GLOBALCONSTANTS byteconst (* Global constants *)
  (* Standard: 61499-1 *)
  (* Version 1.0, 2024-02-22, franz *)
  VAR_GLOBAL CONSTANT
    WORD_BYTE_ZZ : WORD := 16#0000; (* ZERO Constant *)
    WORD_BYTE_00 : WORD := 16#00FF; (* LSB_Byte Constant *)
    WORD_BYTE_01 : WORD := 16#FF00; (* MSB_Byte Constant *)
  END_VAR
END_GLOBALCONSTANTS
